Omron Sysmac Studio project MCS500_V10_2_0_Omron_EIP (Sysmac Studio 1.53.0.64009, StandardProject)
(* Mcs500 V10.2 Demo project EthernetIP *)

# Controller NX1P2_9024DT1: NX1P2-9024DT1 version 1.16
Task PrimaryTask (priority 4, period or condition 2000): MCS500_E001

TYPE MCS500 : STRUCT
    Outputs : Outputs;
    Inputs : Inputs;
    CommandsID : MCS500Cmd;
END_STRUCT END_TYPE
TYPE Inputs : STRUCT
    Status : Status;  (* offset 0.0 *)
    Motion : Motion;  (* offset 4.0 *)
    Joint_Set : Joint_Set;  (* offset 16.0 *)
    EndEffector_Pose : EndEffector_Pose;  (* offset 40.0 *)
    Configurations : Configurations;  (* offset 64.0 *)
    WRF : WRF;  (* offset 68.0 *)
    TRF : TRF;  (* offset 92.0 *)
    TimeStamp : TimeStamp;  (* offset 116.0 *)
    SafetyStatus : SafetyStatus;  (* offset 128.0 *)
    DynamicData0 : DynamicData;  (* offset 140.0 *)
    DynamicData1 : DynamicData;  (* offset 168.0 *)
    DynamicData2 : DynamicData;  (* offset 196.0 *)
    DynamicData3 : DynamicData;  (* offset 224.0 *)
END_STRUCT END_TYPE
TYPE Status : STRUCT  (* Various robot status bits *)
    Busy : BOOL;
    Activated : BOOL;
    Homed : BOOL;
    SimActivated : BOOL;
    BrakesEngaged : BOOL;
    RecoveryMode : BOOL;
    EStop : BOOL;
    CollisionStatus : BOOL;
    WorkzoneStatus : BOOL;
    Error : UINT;  (* Error code (refer to documentation for specific error code meaning) *)
END_STRUCT END_TYPE
TYPE Motion : STRUCT
    CheckPoint : UDINT;  (* Indicates which checkpoint id the robot has reached last; offset 0.0 *)
    MoveID : UINT;  (* Latest move id that was received and queued by the robot; offset 4.0 *)
    FifoSpace : UINT;  (* Number of commands that the robot can receive and queue at the moment; offset 6.0 *)
    Paused : BOOL;  (* offset 8.0 *)
    EOB : BOOL;  (* offset 8.1 *)
    EOM : BOOL;  (* offset 8.2 *)
    FifoCleared : BOOL;  (* offset 8.3 *)
    PStop2 : BOOL;  (* offset 8.4 *)
    ExcessiveTorque : BOOL;  (* offset 8.5 *)
    OfflineProgramID : UINT;  (* Id of the offline program currently running (0 if none); offset 10.0 *)
END_STRUCT END_TYPE
TYPE Joint_Set : STRUCT
    SubIndex001 : REAL;  (* Joint 1's angular position (-140 to +140) *)
    SubIndex002 : REAL;  (* Joint 2's angular position (-145 to +145) *)
    SubIndex003 : REAL;  (* Joint 3's linear position (-102 to 0) *)
    SubIndex004 : REAL;  (* Joint 4's angular position (-3600 to +3600) *)
    SubIndex005 : REAL;  (* Unused on this 4-axes robot *)
    SubIndex006 : REAL;  (* Unused on this 4-axes robot *)
END_STRUCT END_TYPE
TYPE EndEffector_Pose : STRUCT
    SubIndex001 : REAL;  (* X position *)
    SubIndex002 : REAL;  (* Y position *)
    SubIndex003 : REAL;  (* Z position *)
    SubIndex004 : REAL;  (* Alpha-angle position *)
    SubIndex005 : REAL;  (* Beta-angle position *)
    SubIndex006 : REAL;  (* Gamma-angle position *)
END_STRUCT END_TYPE
TYPE Configurations : STRUCT
    Shoulder : SINT;  (* Unused on this 4-axes robot; offset 0.0 *)
    Elbow : SINT;  (* Current elbow inverse kinematics configuration (either -1 or 1); offset 1.0 *)
    Wrist : SINT;  (* Unused on this 4-axes robot; offset 2.0 *)
    Turn : SINT;  (* Current last joint turn (-100 to 100); offset 3.0 *)
END_STRUCT END_TYPE
TYPE WRF : STRUCT
    SubIndex001 : REAL;  (* X position of WRF (relative to BRF) *)
    SubIndex002 : REAL;  (* Y position of WRF (relative to BRF) *)
    SubIndex003 : REAL;  (* Z position of WRF (relative to BRF) *)
    SubIndex004 : REAL;  (* Alpha-angle position of WRF (relative to BRF) *)
    SubIndex005 : REAL;  (* Beta-angle position of WRF (relative to BRF) *)
    SubIndex006 : REAL;  (* Gamma-angle position of WRF (relative to BRF) *)
END_STRUCT END_TYPE
TYPE TRF : STRUCT
    SubIndex001 : REAL;  (* X position of TRF (relative to FRF) *)
    SubIndex002 : REAL;  (* Y position of TRF (relative to FRF) *)
    SubIndex003 : REAL;  (* Z position of TRF (relative to FRF) *)
    SubIndex004 : REAL;  (* Alpha-angle position of TRF (relative to FRF) *)
    SubIndex005 : REAL;  (* Beta-angle position of TRF (relative to FRF) *)
    SubIndex006 : REAL;  (* Gamma-angle position of TRF (relative to FRF) *)
END_STRUCT END_TYPE
TYPE TimeStamp : STRUCT
    Seconds : UDINT;  (* Robot timestamp (seconds) indicating when input info was updated *)
    MicroSeconds : UDINT;  (* Robot timestamp (microsecond part) indicating when input info was updated *)
    DynamicDataCycles : UDINT;  (* Number of times all available dynamic data was updated *)
END_STRUCT END_TYPE
TYPE SafetyStatus : STRUCT
    EStop : BOOL;  (* offset 0.0 *)
    PStop1 : BOOL;  (* offset 0.1 *)
    PStop2 : BOOL;  (* offset 0.2 *)
    OperationModeChange : BOOL;  (* offset 0.4 *)
    EnablingDeviceReleased : BOOL;  (* offset 0.5 *)
    VoltageFluctuation : BOOL;  (* offset 0.6 *)
    Reboot : BOOL;  (* offset 0.7 *)
    RedundancyFault : BOOL;  (* offset 1.0 *)
    StandstillFault : BOOL;  (* offset 1.1 *)
    ConnectionDropped : BOOL;  (* offset 1.2 *)
    MinorError : BOOL;  (* offset 1.3 *)
    EStopResettable : BOOL;  (* offset 4.0 *)
    PStop1Resettable : BOOL;  (* offset 4.1 *)
    PStop2Resettable : BOOL;  (* offset 4.2 *)
    OperationModeChangeResettable : BOOL;  (* offset 4.4 *)
    EnablingDeviceReleasedResettable : BOOL;  (* offset 4.5 *)
    VolatgeFluctuationResettable : BOOL;  (* offset 4.6 *)
    RebootResettable : BOOL;  (* offset 4.7 *)
    RedundancyFaultResettable : BOOL;  (* offset 5.0 *)
    StandstillFaultResettable : BOOL;  (* offset 5.1 *)
    ConnectionDroppedResettable : BOOL;  (* offset 5.2 *)
    MinorErrorResettable : BOOL;  (* offset 5.3 *)
    OperationMode : SINT;  (* offset 8.0 *)
    ResetReady : BOOL;  (* offset 9.0 *)
    VMotorOn : BOOL;  (* offset 9.1 *)
    PowerSupplyInput_EStop : BOOL;  (* offset 9.2 *)
    PowerSupplyInput_PStop1 : BOOL;  (* offset 9.3 *)
    PowerSupplyInput_PStop2 : BOOL;  (* offset 9.4 *)
    PowerSupplyInput_External : BOOL;  (* offset 9.5 *)
    PowerSupplyInput_Keypad : BOOL;  (* offset 9.6 *)
    PowerSupplyInput_Enabling : BOOL;  (* offset 9.7 *)
END_STRUCT END_TYPE
TYPE DynamicData : STRUCT
    DynamicDataType : UDINT;  (* Dynamic type of the 6 following values *)
    DynamicDataValue0 : REAL;
    DynamicDataValue1 : REAL;
    DynamicDataValue2 : REAL;
    DynamicDataValue3 : REAL;
    DynamicDataValue4 : REAL;
    DynamicDataValue5 : REAL;
END_STRUCT END_TYPE
TYPE Outputs : STRUCT
    RobotControl : RobotControl;  (* offset 0.0 *)
    MotionControl : MotionControl;  (* offset 4.0 *)
    MotionCommand : MotionCommand;  (* offset 8.0 *)
    HostTime : UDINT;  (* Host absolute time in seconds since epoch (to synchronize robot's time); offset 36.0 *)
    BrakesControlAllowed : BOOL;  (* offset 40.0 *)
    BrakesEngaged : BOOL;  (* offset 40.1 *)
    DynamicDataCfg0 : UDINT;  (* Type of dynamic data to return in dynamic data index 0; offset 44.0 *)
    DynamicDataCfg1 : UDINT;  (* Type of dynamic data to return in dynamic data index 1; offset 48.0 *)
    DynamicDataCfg2 : UDINT;  (* Type of dynamic data to return in dynamic data index 2; offset 52.0 *)
    DynamicDataCfg3 : UDINT;  (* Type of dynamic data to return in dynamic data index 3; offset 56.0 *)
END_STRUCT END_TYPE
TYPE RobotControl : STRUCT  (* Various robot control bits *)
    Deactivate : BOOL;  (* offset 0.0 *)
    Activate : BOOL;  (* offset 0.1 *)
    Home : BOOL;  (* offset 0.2 *)
    ResetError : BOOL;  (* offset 0.3 *)
    EnableSimulation : BOOL;  (* offset 0.4 *)
    EnableRecoveryMode : BOOL;  (* offset 0.5 *)
    DisableEtherCAT : BOOL;  (* offset 0.6 *)
END_STRUCT END_TYPE
TYPE MotionControl : STRUCT  (* Various motion control bits *)
    MoveID : UINT;  (* User-defined id of the command currently being sent (The robot will consider a new command is sent only when moveId is changed); offset 0.0 *)
    Setpoint : BOOL;  (* offset 2.0 *)
    PauseMotion : BOOL;  (* offset 2.1 *)
    ClearMotion : BOOL;  (* offset 2.2 *)
    ResumeMotion : BOOL;  (* offset 2.3 *)
END_STRUCT END_TYPE
TYPE MotionCommand : STRUCT
    MoveCommand : UDINT;  (* The move command to apply; offset 0.0 *)
    MoveSubIndex001 : REAL;  (* Argument 1 for move command; offset 4.0 *)
    MoveSubIndex002 : REAL;  (* Argument 2 for move command; offset 8.0 *)
    MoveSubIndex003 : REAL;  (* Argument 3 for move command; offset 12.0 *)
    MoveSubIndex004 : REAL;  (* Argument 4 for move command; offset 16.0 *)
    MoveSubIndex005 : REAL;  (* Argument 5 for move command; offset 20.0 *)
    MoveSubIndex006 : REAL;  (* Argument 6 for move command; offset 24.0 *)
END_STRUCT END_TYPE
TYPE MCS500Cmd : (NoCmd := 00, MoveJoints := 01, MovePose := 02, MoveLin := 03, MoveLinRelTrf := 04, MoveLinRelWrf := 05, Delay := 06, SetBlending := 07, SetJointVel := 08, SetJointAcc := 09, SetCartAngVel := 10, SetCartLinVel := 11, SetCartAcc := 12, SetTrf := 13, SetWrf := 14, SetConf := 15, SetAutoConf := 16, SetCheckpoint := 17, MoveJointsVel := 21, MoveLinVelWrf := 22, MoveLinVelTrf := 23, SetVelTimeout := 24, SetConfTurn := 25, SetAutoConfTurn := 26, SetTorqueLimits := 27, SetTorquesLimitCfg := 28, MoveJointsRel := 29, SetJointVelLimit := 33, SetOutputState := 34, SetOutputState_Immediate := 35, SetIoSim := 36, VacuumGrip := 37, VacuumGrip_Immediate := 38, VacuumRelease := 39, VacuumRelease_Immediate := 40, SetVacuumThreshold := 41, SetVacuumThreshold_Immediate := 42, SetVacuumPurgeDuration := 43, SetVacuumPurgeDuration_Immediate := 44, MoveJump := 45, SetMoveJumpHeight := 46, SetMoveJumpApproachVel := 47, SetTimeScaling := 48, StartProgram := 100); END_TYPE

VAR_GLOBAL
    E001 : MCS500;  (* Robot Structure				PLC *)
    E001_Inputs : Inputs;  (* EthernetIp Inputs				PLC; network input *)
    E001_Outputs : Outputs;  (* EthernetIP Outputs				PLC; network output *)
END_VAR

PROGRAM MCS500_E001
VAR
    Activate : BOOL;
    Deactivate : BOOL;
    Home : BOOL;
    ResetError : BOOL;
    Pause : BOOL;
    RecoveryMode : BOOL;
    StartSequence : BOOL;
    SetCheckpoint1Buffered : BOOL;
    ExecuteMove : BOOL;
    SetCartLinVel1Buffered : BOOL;
    MovePose1Buffered : BOOL;
    SetCartLinVel1 : MCS500_SetCartLinVel;
    MovePose1 : MCS500_MovePose;
    SetCheckpoint1 : MCS500_SetCheckpoint;
    Argument : ARRAY[0..5] OF real;  (* Array for positions *)
    StepSquareMove : INT;  (* Sequencer step *)
    SetJointsVel1 : MCS500_SetJointsVel;
    SetJointsVel1Buffered : BOOL;
    ResumeMotion : BOOL;
    SetTrf1 : MCS500_SetTrf;
    SetTrf1Buffered : BOOL;
    SetWrf1 : MCS500_SetWrf;
    SetBlending1 : MCS500_SetBlending;
    SetBlending1Buffered : BOOL;
    SetConf1 : MCS500_SetConf;
    MoveLin1 : MCS500_MoveLin;
    MoveLin1Buffered : BOOL;
    SetMoveJumpApproachVel1 : MCS500_SetMoveJumpApproachVel;
    SetMoveJumpApproachVel1Buffered : BOOL;
    SetMoveJumpHeight1 : MCS500_SetMoveJumpHeight;
    SetMoveJumpHeight1Buffered : BOOL;
    MoveJump1 : MCS500_MoveJump;
    MoveJump1Buffered : BOOL;
    SetConf1Buffered : BOOL;
    E002 : MCS500;
    SetWrf1Buffered : BOOL;
    Delay1 : MCS500_Delay;
    Delay1Buffered : BOOL;
    SimulationMode : BOOL;
    ResetSequence : BOOL;
    IOModuleInfo : DWORD;
    IOModuleOutputsValues : DWORD;
    IOModuleInputsValues : DWORD;
    IOModuleSimMode : BOOL;
    IOModulePresent : BOOL;
    IOModuleErrorCode : BYTE;
    IOModuleNbInput : BYTE;
    IOModuleNbOutput : BYTE;
END_VAR
VAR_EXTERNAL
    E001_Inputs : Inputs;
    E001_Outputs : Outputs;
    E001 : MCS500;
END_VAR
VAR
    _e1 : R_TRIG;
END_VAR

(* Section IOs: ladder, written here as Structured Text *)

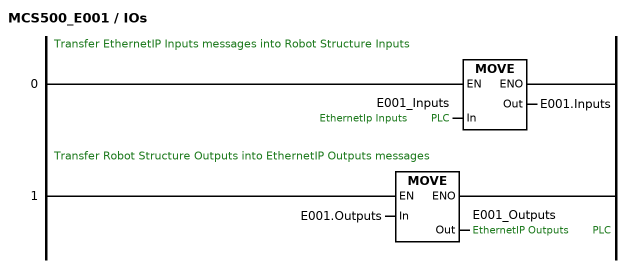
(* Rung 0: Transfer EthernetIP Inputs messages into Robot Structure Inputs *)
E001.Inputs := E001_Inputs;
(* Rung 1: Transfer Robot Structure Outputs into EthernetIP Outputs messages *)
E001_Outputs := E001.Outputs;

(* Section Robot_Control: ladder, written here as Structured Text *)

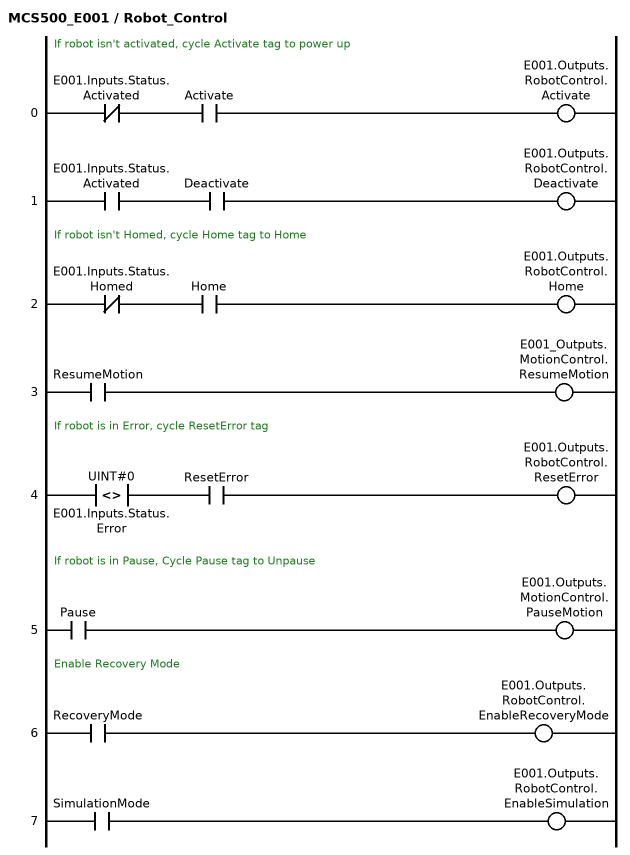
(* Rung 0: If robot isn't activated, cycle Activate tag to power up *)
E001.Outputs.RobotControl.Activate := NOT E001.Inputs.Status.Activated AND Activate;
(* Rung 1 *)
E001.Outputs.RobotControl.Deactivate := E001.Inputs.Status.Activated AND Deactivate;
(* Rung 2: If robot isn't Homed, cycle Home tag to Home *)
E001.Outputs.RobotControl.Home := NOT E001.Inputs.Status.Homed AND Home;
(* Rung 3 *)
E001_Outputs.MotionControl.ResumeMotion := ResumeMotion;
(* Rung 4: If robot is in Error, cycle ResetError tag *)
E001.Outputs.RobotControl.ResetError := (UINT#0 <> E001.Inputs.Status.Error) AND ResetError;
(* Rung 5: If robot is in Pause, Cycle Pause tag to Unpause *)
E001.Outputs.MotionControl.PauseMotion := Pause;
(* Rung 6: Enable Recovery Mode *)
E001.Outputs.RobotControl.EnableRecoveryMode := RecoveryMode;
(* Rung 7 *)
E001.Outputs.RobotControl.EnableSimulation := SimulationMode;

(* Section Sequence: ladder, written here as Structured Text *)

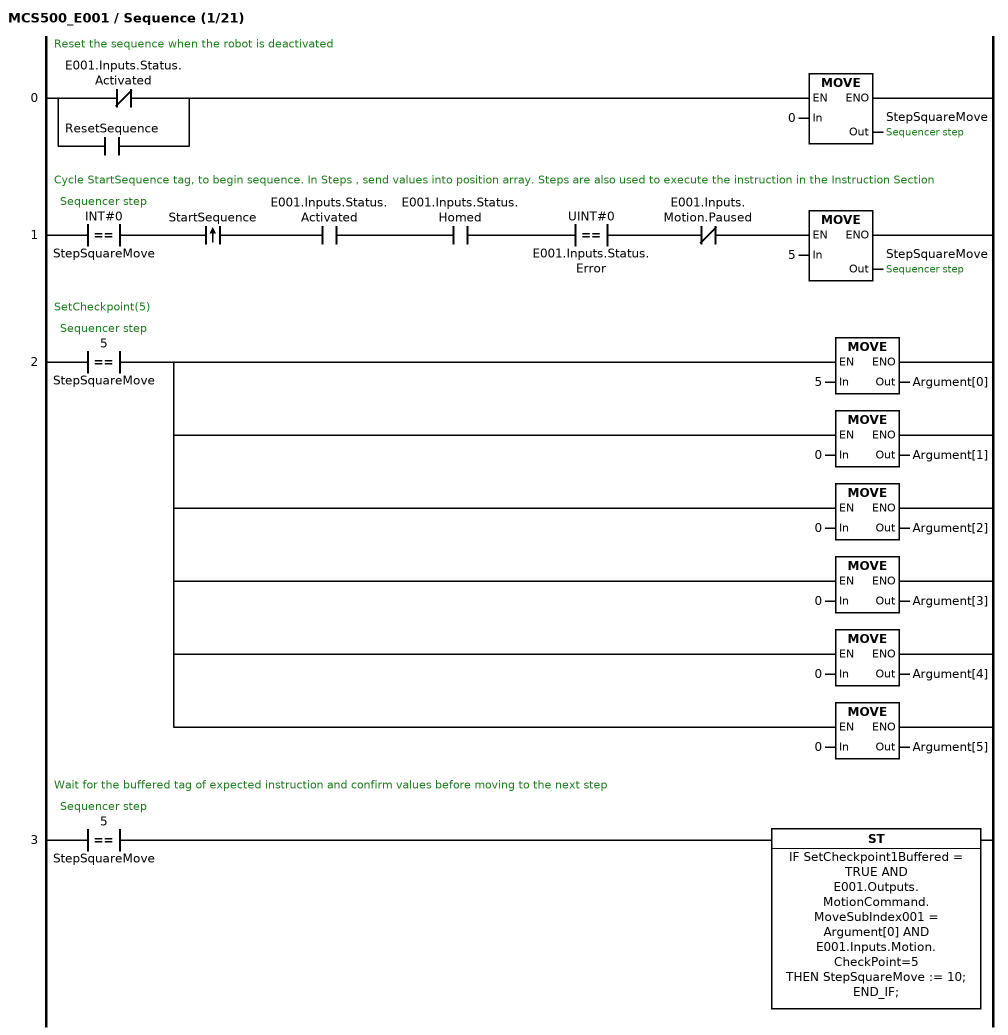
(* Rung 0: Reset the sequence when the robot is deactivated *)
IF NOT E001.Inputs.Status.Activated OR ResetSequence THEN StepSquareMove := 0; END_IF;
(* Rung 1: Cycle StartSequence tag, to begin sequence. In Steps , send values into position array. Steps are also used to execute the instruction in the Instruction Section *)
_e1(CLK := StartSequence);
IF (INT#0 = StepSquareMove) AND _e1.Q AND E001.Inputs.Status.Activated AND E001.Inputs.Status.Homed AND (UINT#0 = E001.Inputs.Status.Error) AND NOT E001.Inputs.Motion.Paused THEN
    StepSquareMove := 5;
END_IF;
(* Rung 2: SetCheckpoint(5) *)
IF 5 = StepSquareMove THEN
    Argument[0] := 5;
    Argument[1] := 0;
    Argument[2] := 0;
    Argument[3] := 0;
    Argument[4] := 0;
    Argument[5] := 0;
END_IF;
(* Rung 3: Wait for the buffered tag of expected instruction and confirm values before moving to the next step *)
IF 5 = StepSquareMove THEN
    IF SetCheckpoint1Buffered = TRUE AND
    	E001.Outputs.MotionCommand.MoveSubIndex001 = Argument[0] AND
    	E001.Inputs.Motion.CheckPoint=5
    	THEN StepSquareMove := 10;
    END_IF;
END_IF;

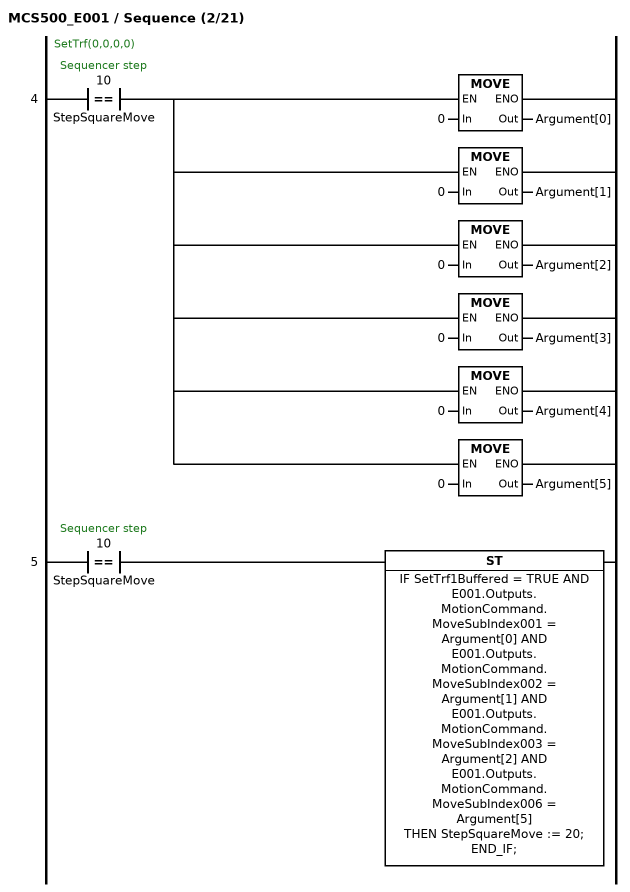
(* Rung 4: SetTrf(0,0,0,0) *)
IF 10 = StepSquareMove THEN
    Argument[0] := 0;
    Argument[1] := 0;
    Argument[2] := 0;
    Argument[3] := 0;
    Argument[4] := 0;
    Argument[5] := 0;
END_IF;
(* Rung 5 *)
IF 10 = StepSquareMove THEN
    IF SetTrf1Buffered = TRUE AND
    	E001.Outputs.MotionCommand.MoveSubIndex001 = Argument[0] AND
    	E001.Outputs.MotionCommand.MoveSubIndex002 = Argument[1] AND
    	E001.Outputs.MotionCommand.MoveSubIndex003 = Argument[2] AND
    	E001.Outputs.MotionCommand.MoveSubIndex006 = Argument[5] 
    	THEN StepSquareMove := 20;
    END_IF;
END_IF;

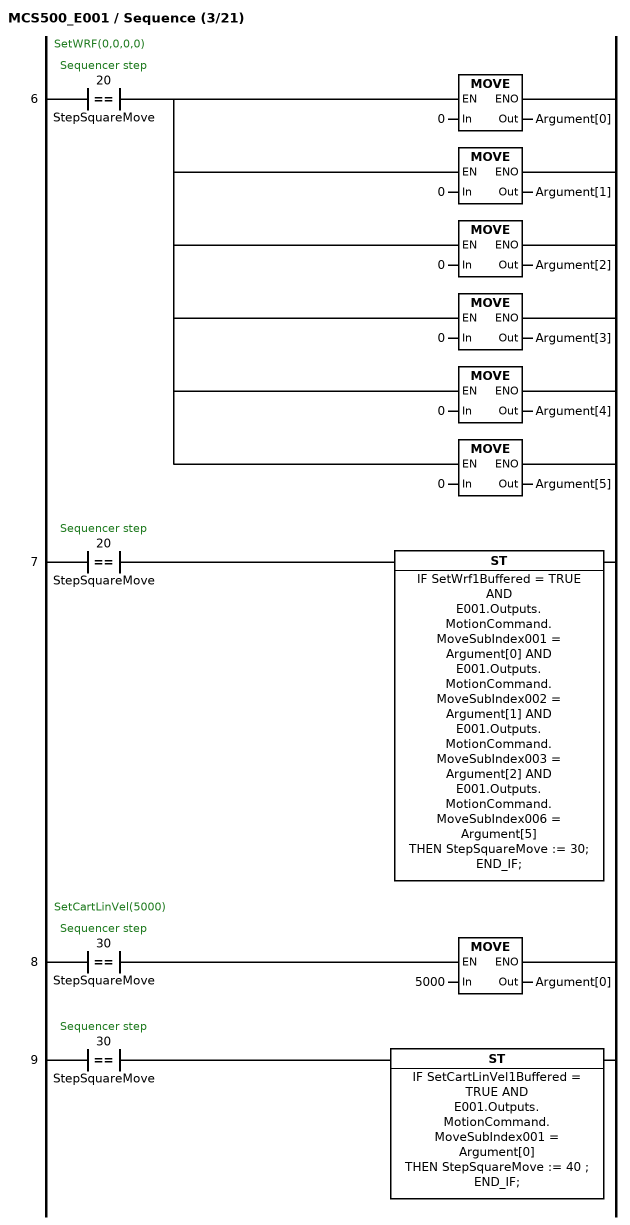
(* Rung 6: SetWRF(0,0,0,0) *)
IF 20 = StepSquareMove THEN
    Argument[0] := 0;
    Argument[1] := 0;
    Argument[2] := 0;
    Argument[3] := 0;
    Argument[4] := 0;
    Argument[5] := 0;
END_IF;
(* Rung 7 *)
IF 20 = StepSquareMove THEN
    IF SetWrf1Buffered = TRUE AND
    	E001.Outputs.MotionCommand.MoveSubIndex001 = Argument[0] AND
    	E001.Outputs.MotionCommand.MoveSubIndex002 = Argument[1] AND
    	E001.Outputs.MotionCommand.MoveSubIndex003 = Argument[2] AND
    	E001.Outputs.MotionCommand.MoveSubIndex006 = Argument[5] 
    	THEN StepSquareMove := 30;
    END_IF;
END_IF;
(* Rung 8: SetCartLinVel(5000) *)
IF 30 = StepSquareMove THEN Argument[0] := 5000; END_IF;
(* Rung 9 *)
IF 30 = StepSquareMove THEN
    IF SetCartLinVel1Buffered = TRUE AND
    	E001.Outputs.MotionCommand.MoveSubIndex001 = Argument[0] 
    	THEN StepSquareMove := 40 ;
    END_IF;
END_IF;

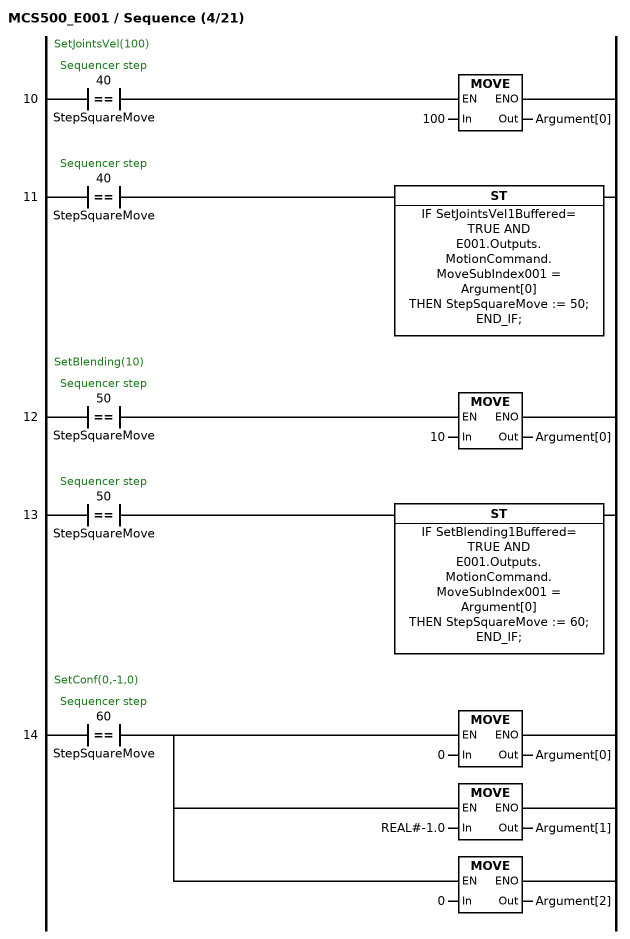
(* Rung 10: SetJointsVel(100) *)
IF 40 = StepSquareMove THEN Argument[0] := 100; END_IF;
(* Rung 11 *)
IF 40 = StepSquareMove THEN
    IF SetJointsVel1Buffered= TRUE AND
    	E001.Outputs.MotionCommand.MoveSubIndex001 = Argument[0]
    	THEN StepSquareMove := 50;
    END_IF;
END_IF;
(* Rung 12: SetBlending(10) *)
IF 50 = StepSquareMove THEN Argument[0] := 10; END_IF;
(* Rung 13 *)
IF 50 = StepSquareMove THEN
    IF SetBlending1Buffered= TRUE AND
    	E001.Outputs.MotionCommand.MoveSubIndex001 = Argument[0]
    	THEN StepSquareMove := 60;
    END_IF;
END_IF;
(* Rung 14: SetConf(0,-1,0) *)
IF 60 = StepSquareMove THEN
    Argument[0] := 0;
    Argument[1] := REAL#-1.0;
    Argument[2] := 0;
END_IF;

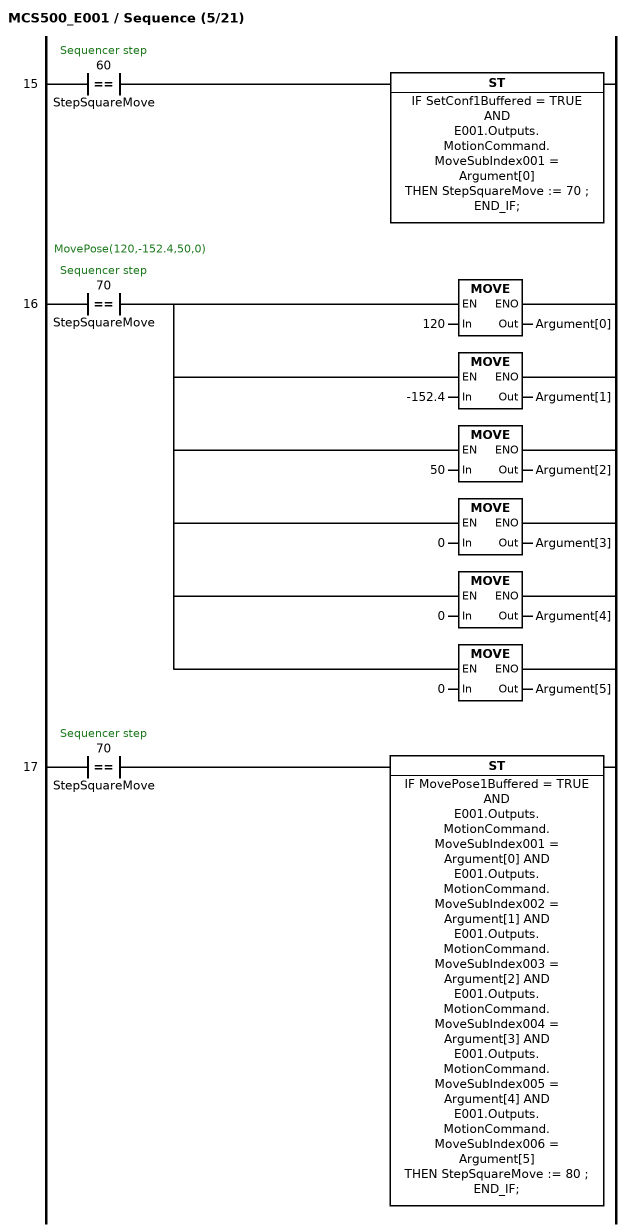
(* Rung 15 *)
IF 60 = StepSquareMove THEN
    IF SetConf1Buffered = TRUE AND
    	E001.Outputs.MotionCommand.MoveSubIndex001 = Argument[0]
    	THEN StepSquareMove := 70 ;
    END_IF;
END_IF;
(* Rung 16: MovePose(120,-152.4,50,0) *)
IF 70 = StepSquareMove THEN
    Argument[0] := 120;
    Argument[1] := -152.4;
    Argument[2] := 50;
    Argument[3] := 0;
    Argument[4] := 0;
    Argument[5] := 0;
END_IF;
(* Rung 17 *)
IF 70 = StepSquareMove THEN
    IF MovePose1Buffered = TRUE AND
    	E001.Outputs.MotionCommand.MoveSubIndex001 = Argument[0] AND
    	E001.Outputs.MotionCommand.MoveSubIndex002 = Argument[1] AND
    	E001.Outputs.MotionCommand.MoveSubIndex003 = Argument[2] AND
    	E001.Outputs.MotionCommand.MoveSubIndex004 = Argument[3] AND
    	E001.Outputs.MotionCommand.MoveSubIndex005 = Argument[4] AND
    	E001.Outputs.MotionCommand.MoveSubIndex006 = Argument[5] 
    	THEN StepSquareMove := 80 ;
    END_IF;
END_IF;

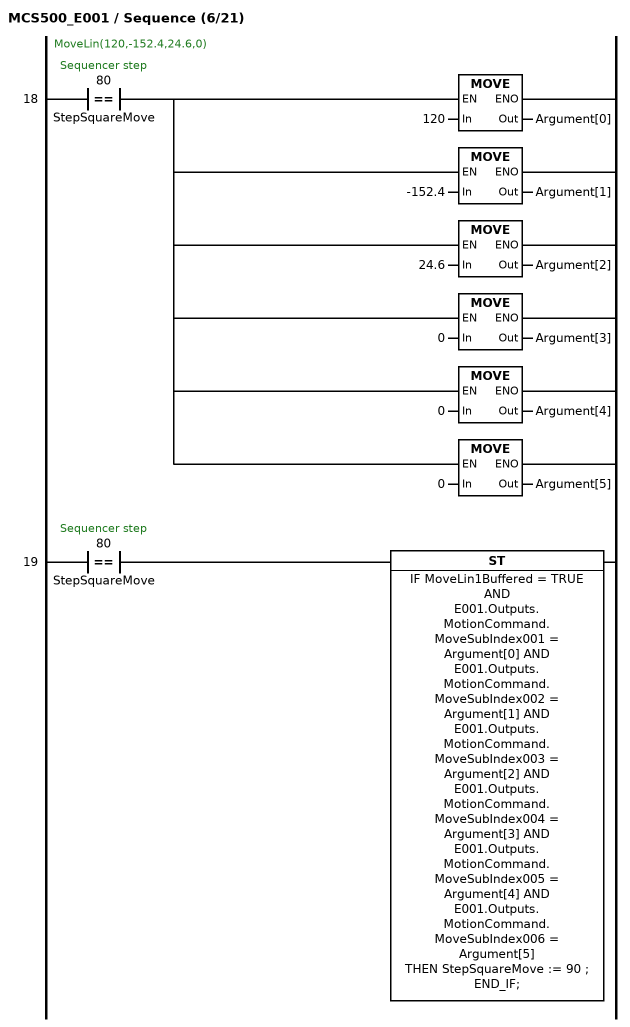
(* Rung 18: MoveLin(120,-152.4,24.6,0) *)
IF 80 = StepSquareMove THEN
    Argument[0] := 120;
    Argument[1] := -152.4;
    Argument[2] := 24.6;
    Argument[3] := 0;
    Argument[4] := 0;
    Argument[5] := 0;
END_IF;
(* Rung 19 *)
IF 80 = StepSquareMove THEN
    IF MoveLin1Buffered = TRUE AND
    	E001.Outputs.MotionCommand.MoveSubIndex001 = Argument[0] AND
    	E001.Outputs.MotionCommand.MoveSubIndex002 = Argument[1] AND
    	E001.Outputs.MotionCommand.MoveSubIndex003 = Argument[2] AND
    	E001.Outputs.MotionCommand.MoveSubIndex004 = Argument[3] AND
    	E001.Outputs.MotionCommand.MoveSubIndex005 = Argument[4] AND
    	E001.Outputs.MotionCommand.MoveSubIndex006 = Argument[5] 
    	THEN StepSquareMove := 90 ;
    END_IF;
END_IF;

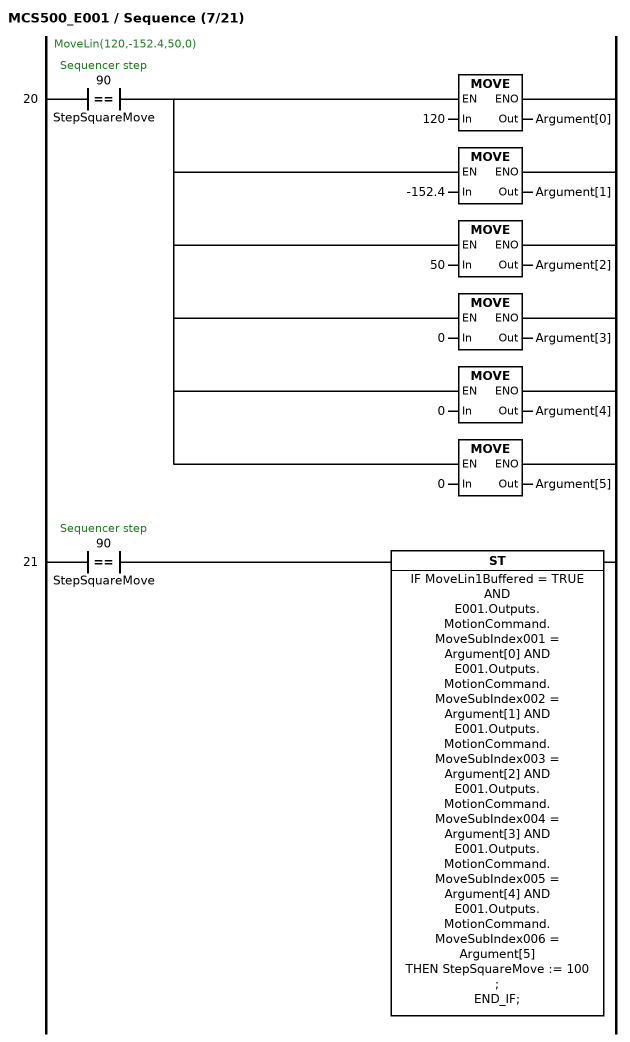
(* Rung 20: MoveLin(120,-152.4,50,0) *)
IF 90 = StepSquareMove THEN
    Argument[0] := 120;
    Argument[1] := -152.4;
    Argument[2] := 50;
    Argument[3] := 0;
    Argument[4] := 0;
    Argument[5] := 0;
END_IF;
(* Rung 21 *)
IF 90 = StepSquareMove THEN
    IF MoveLin1Buffered = TRUE AND
    	E001.Outputs.MotionCommand.MoveSubIndex001 = Argument[0] AND
    	E001.Outputs.MotionCommand.MoveSubIndex002 = Argument[1] AND
    	E001.Outputs.MotionCommand.MoveSubIndex003 = Argument[2] AND
    	E001.Outputs.MotionCommand.MoveSubIndex004 = Argument[3] AND
    	E001.Outputs.MotionCommand.MoveSubIndex005 = Argument[4] AND
    	E001.Outputs.MotionCommand.MoveSubIndex006 = Argument[5] 
    	THEN StepSquareMove := 100 ;
    END_IF;
END_IF;

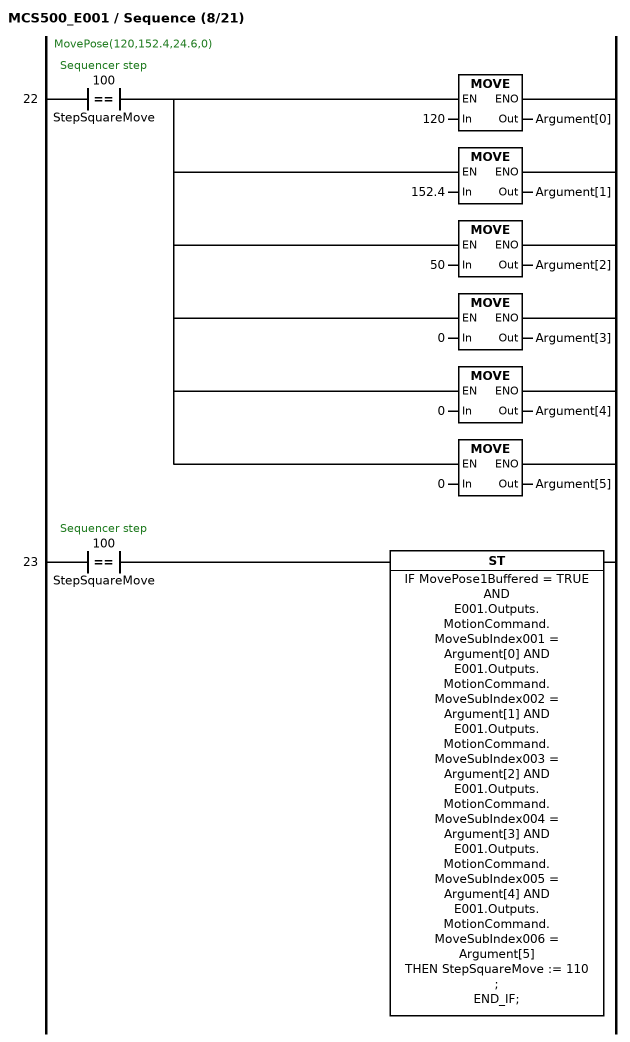
(* Rung 22: MovePose(120,152.4,24.6,0) *)
IF 100 = StepSquareMove THEN
    Argument[0] := 120;
    Argument[1] := 152.4;
    Argument[2] := 50;
    Argument[3] := 0;
    Argument[4] := 0;
    Argument[5] := 0;
END_IF;
(* Rung 23 *)
IF 100 = StepSquareMove THEN
    IF MovePose1Buffered = TRUE AND
    	E001.Outputs.MotionCommand.MoveSubIndex001 = Argument[0] AND
    	E001.Outputs.MotionCommand.MoveSubIndex002 = Argument[1] AND
    	E001.Outputs.MotionCommand.MoveSubIndex003 = Argument[2] AND
    	E001.Outputs.MotionCommand.MoveSubIndex004 = Argument[3] AND
    	E001.Outputs.MotionCommand.MoveSubIndex005 = Argument[4] AND
    	E001.Outputs.MotionCommand.MoveSubIndex006 = Argument[5] 
    	THEN StepSquareMove := 110 ;
    END_IF;
END_IF;

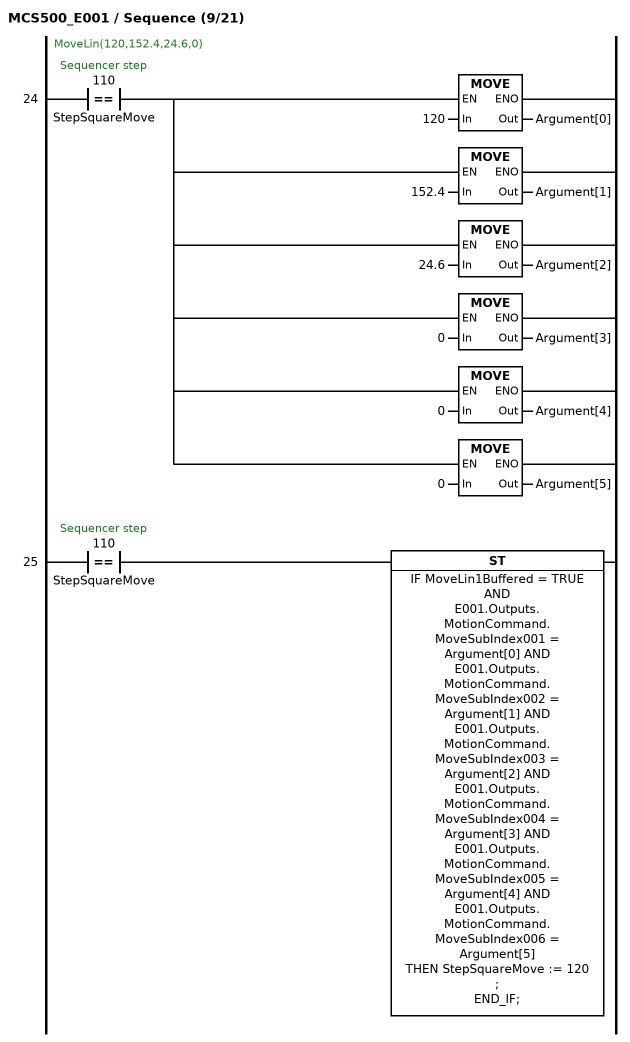
(* Rung 24: MoveLin(120,152.4,24.6,0) *)
IF 110 = StepSquareMove THEN
    Argument[0] := 120;
    Argument[1] := 152.4;
    Argument[2] := 24.6;
    Argument[3] := 0;
    Argument[4] := 0;
    Argument[5] := 0;
END_IF;
(* Rung 25 *)
IF 110 = StepSquareMove THEN
    IF MoveLin1Buffered = TRUE AND
    	E001.Outputs.MotionCommand.MoveSubIndex001 = Argument[0] AND
    	E001.Outputs.MotionCommand.MoveSubIndex002 = Argument[1] AND
    	E001.Outputs.MotionCommand.MoveSubIndex003 = Argument[2] AND
    	E001.Outputs.MotionCommand.MoveSubIndex004 = Argument[3] AND
    	E001.Outputs.MotionCommand.MoveSubIndex005 = Argument[4] AND
    	E001.Outputs.MotionCommand.MoveSubIndex006 = Argument[5] 
    	THEN StepSquareMove := 120 ;
    END_IF;
END_IF;

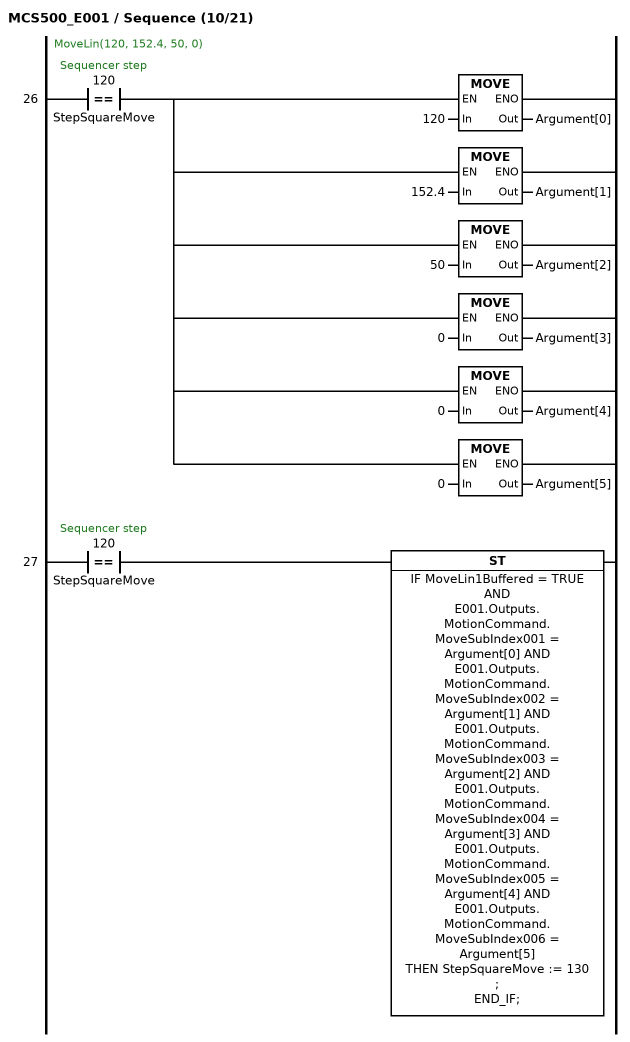
(* Rung 26: MoveLin(120, 152.4, 50, 0) *)
IF 120 = StepSquareMove THEN
    Argument[0] := 120;
    Argument[1] := 152.4;
    Argument[2] := 50;
    Argument[3] := 0;
    Argument[4] := 0;
    Argument[5] := 0;
END_IF;
(* Rung 27 *)
IF 120 = StepSquareMove THEN
    IF MoveLin1Buffered = TRUE AND
    	E001.Outputs.MotionCommand.MoveSubIndex001 = Argument[0] AND
    	E001.Outputs.MotionCommand.MoveSubIndex002 = Argument[1] AND
    	E001.Outputs.MotionCommand.MoveSubIndex003 = Argument[2] AND
    	E001.Outputs.MotionCommand.MoveSubIndex004 = Argument[3] AND
    	E001.Outputs.MotionCommand.MoveSubIndex005 = Argument[4] AND
    	E001.Outputs.MotionCommand.MoveSubIndex006 = Argument[5] 
    	THEN StepSquareMove := 130 ;
    END_IF;
END_IF;

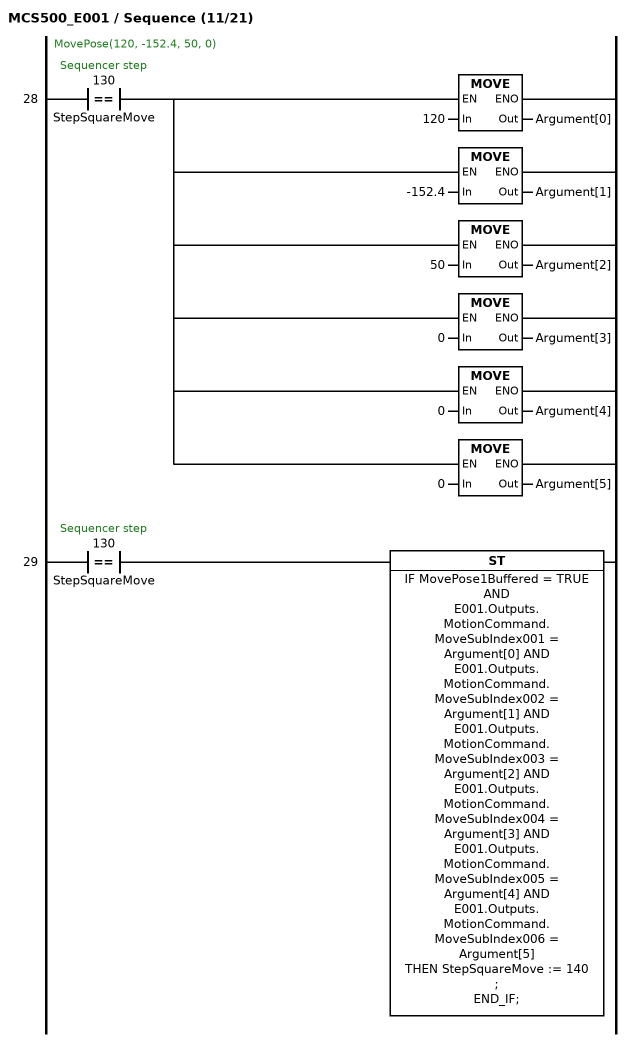
(* Rung 28: MovePose(120, -152.4, 50, 0) *)
IF 130 = StepSquareMove THEN
    Argument[0] := 120;
    Argument[1] := -152.4;
    Argument[2] := 50;
    Argument[3] := 0;
    Argument[4] := 0;
    Argument[5] := 0;
END_IF;
(* Rung 29 *)
IF 130 = StepSquareMove THEN
    IF MovePose1Buffered = TRUE AND
    	E001.Outputs.MotionCommand.MoveSubIndex001 = Argument[0] AND
    	E001.Outputs.MotionCommand.MoveSubIndex002 = Argument[1] AND
    	E001.Outputs.MotionCommand.MoveSubIndex003 = Argument[2] AND
    	E001.Outputs.MotionCommand.MoveSubIndex004 = Argument[3] AND
    	E001.Outputs.MotionCommand.MoveSubIndex005 = Argument[4] AND
    	E001.Outputs.MotionCommand.MoveSubIndex006 = Argument[5] 
    	THEN StepSquareMove := 140 ;
    END_IF;
END_IF;

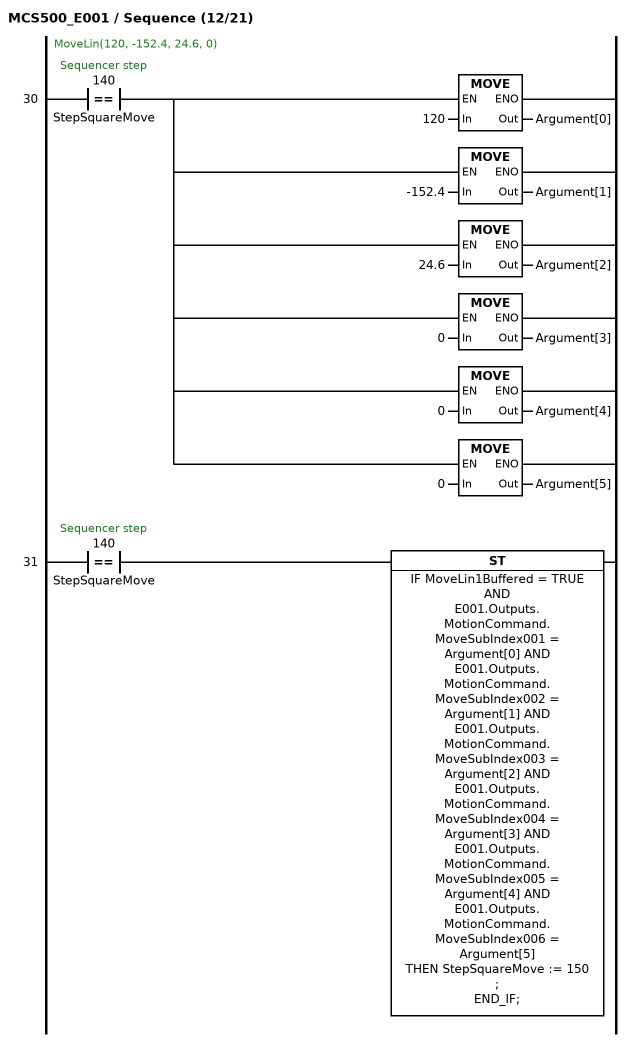
(* Rung 30: MoveLin(120, -152.4, 24.6, 0) *)
IF 140 = StepSquareMove THEN
    Argument[0] := 120;
    Argument[1] := -152.4;
    Argument[2] := 24.6;
    Argument[3] := 0;
    Argument[4] := 0;
    Argument[5] := 0;
END_IF;
(* Rung 31 *)
IF 140 = StepSquareMove THEN
    IF MoveLin1Buffered = TRUE AND
    	E001.Outputs.MotionCommand.MoveSubIndex001 = Argument[0] AND
    	E001.Outputs.MotionCommand.MoveSubIndex002 = Argument[1] AND
    	E001.Outputs.MotionCommand.MoveSubIndex003 = Argument[2] AND
    	E001.Outputs.MotionCommand.MoveSubIndex004 = Argument[3] AND
    	E001.Outputs.MotionCommand.MoveSubIndex005 = Argument[4] AND
    	E001.Outputs.MotionCommand.MoveSubIndex006 = Argument[5] 
    	THEN StepSquareMove := 150 ;
    END_IF;
END_IF;

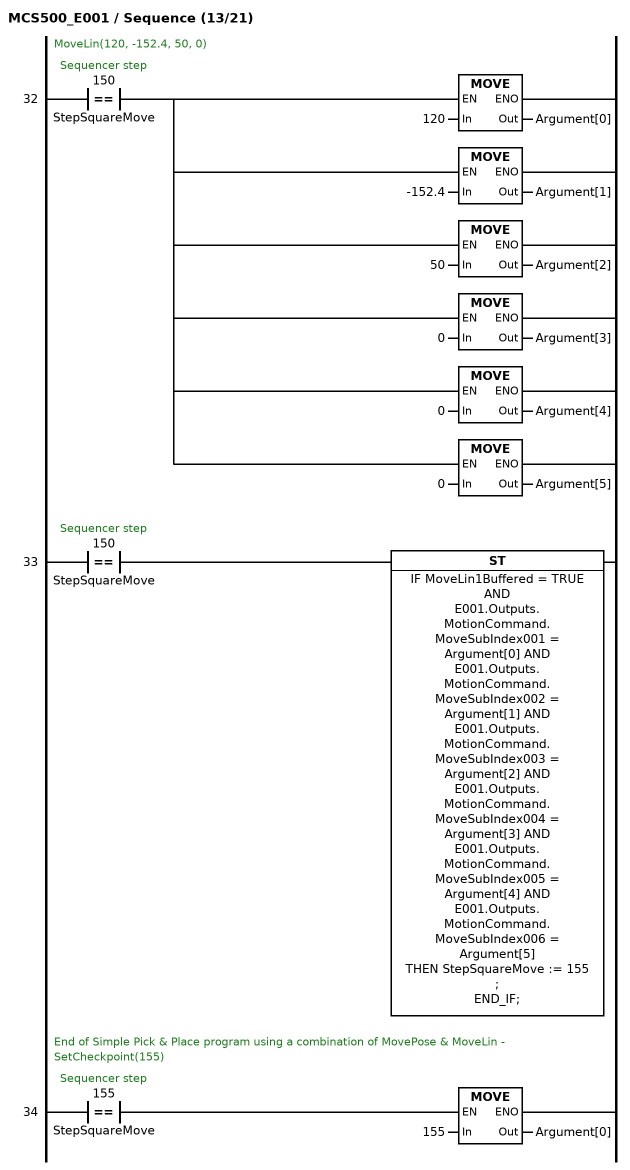
(* Rung 32: MoveLin(120, -152.4, 50, 0) *)
IF 150 = StepSquareMove THEN
    Argument[0] := 120;
    Argument[1] := -152.4;
    Argument[2] := 50;
    Argument[3] := 0;
    Argument[4] := 0;
    Argument[5] := 0;
END_IF;
(* Rung 33 *)
IF 150 = StepSquareMove THEN
    IF MoveLin1Buffered = TRUE AND
    	E001.Outputs.MotionCommand.MoveSubIndex001 = Argument[0] AND
    	E001.Outputs.MotionCommand.MoveSubIndex002 = Argument[1] AND
    	E001.Outputs.MotionCommand.MoveSubIndex003 = Argument[2] AND
    	E001.Outputs.MotionCommand.MoveSubIndex004 = Argument[3] AND
    	E001.Outputs.MotionCommand.MoveSubIndex005 = Argument[4] AND
    	E001.Outputs.MotionCommand.MoveSubIndex006 = Argument[5] 
    	THEN StepSquareMove := 155 ;
    END_IF;
END_IF;
(* Rung 34: End of Simple Pick & Place program using a combination of MovePose & MoveLin - SetCheckpoint(155) *)
IF 155 = StepSquareMove THEN Argument[0] := 155; END_IF;

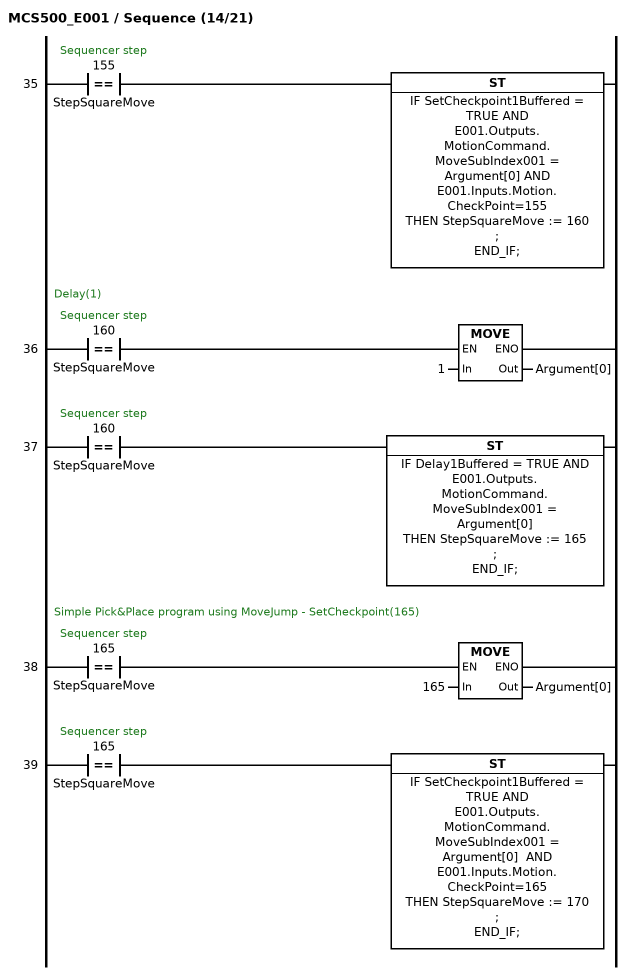
(* Rung 35 *)
IF 155 = StepSquareMove THEN
    IF SetCheckpoint1Buffered = TRUE AND
    	E001.Outputs.MotionCommand.MoveSubIndex001 = Argument[0] AND
    	E001.Inputs.Motion.CheckPoint=155
    	THEN StepSquareMove := 160 ;
    END_IF;
END_IF;
(* Rung 36: Delay(1) *)
IF 160 = StepSquareMove THEN Argument[0] := 1; END_IF;
(* Rung 37 *)
IF 160 = StepSquareMove THEN
    IF Delay1Buffered = TRUE AND
    	E001.Outputs.MotionCommand.MoveSubIndex001 = Argument[0]  
    	THEN StepSquareMove := 165 ;
    END_IF;
END_IF;
(* Rung 38: Simple Pick&Place program using MoveJump - SetCheckpoint(165) *)
IF 165 = StepSquareMove THEN Argument[0] := 165; END_IF;
(* Rung 39 *)
IF 165 = StepSquareMove THEN
    IF SetCheckpoint1Buffered = TRUE AND
    	E001.Outputs.MotionCommand.MoveSubIndex001 = Argument[0]  AND
    	E001.Inputs.Motion.CheckPoint=165
    	THEN StepSquareMove := 170 ;
    END_IF;
END_IF;

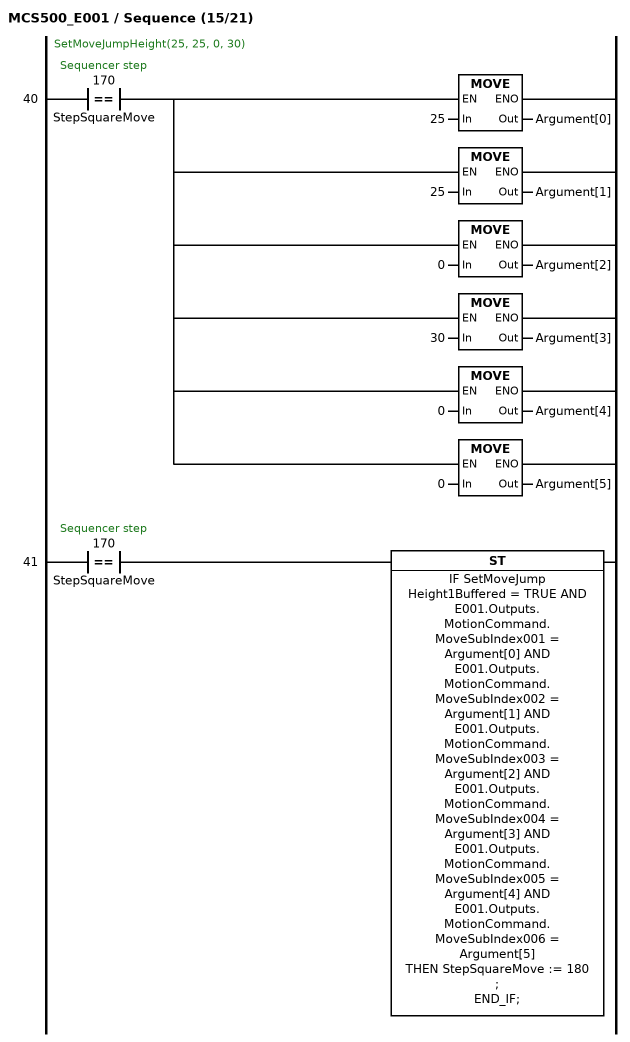
(* Rung 40: SetMoveJumpHeight(25, 25, 0, 30) *)
IF 170 = StepSquareMove THEN
    Argument[0] := 25;
    Argument[1] := 25;
    Argument[2] := 0;
    Argument[3] := 30;
    Argument[4] := 0;
    Argument[5] := 0;
END_IF;
(* Rung 41 *)
IF 170 = StepSquareMove THEN
    IF SetMoveJumpHeight1Buffered = TRUE AND
    	E001.Outputs.MotionCommand.MoveSubIndex001 = Argument[0] AND
    	E001.Outputs.MotionCommand.MoveSubIndex002 = Argument[1] AND
    	E001.Outputs.MotionCommand.MoveSubIndex003 = Argument[2] AND
    	E001.Outputs.MotionCommand.MoveSubIndex004 = Argument[3] AND
    	E001.Outputs.MotionCommand.MoveSubIndex005 = Argument[4] AND
    	E001.Outputs.MotionCommand.MoveSubIndex006 = Argument[5] 
    	THEN StepSquareMove := 180 ;
    END_IF;
END_IF;

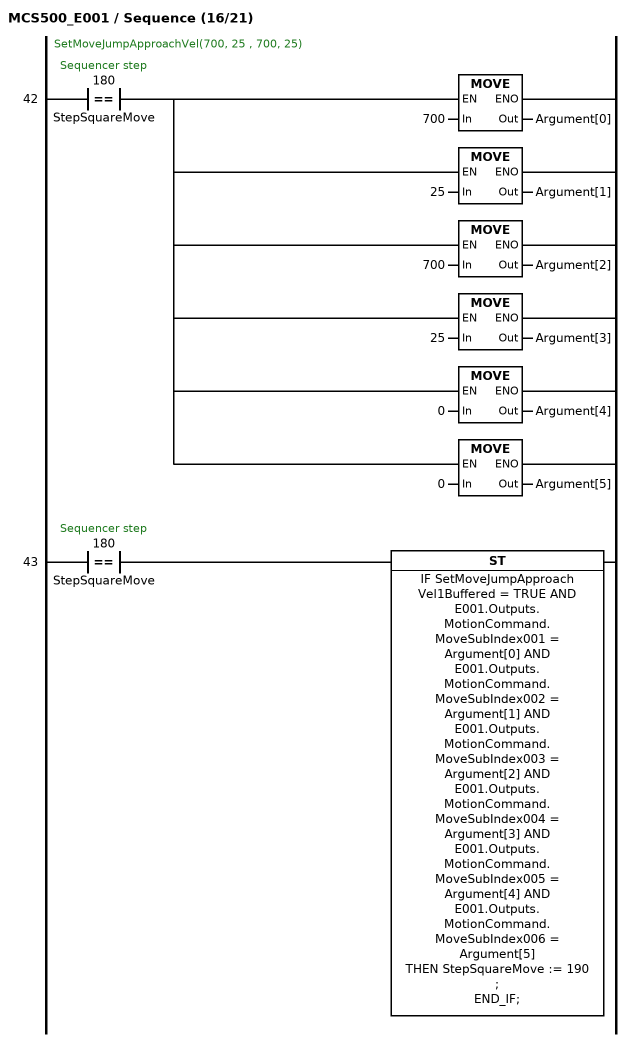
(* Rung 42: SetMoveJumpApproachVel(700, 25 , 700, 25) *)
IF 180 = StepSquareMove THEN
    Argument[0] := 700;
    Argument[1] := 25;
    Argument[2] := 700;
    Argument[3] := 25;
    Argument[4] := 0;
    Argument[5] := 0;
END_IF;
(* Rung 43 *)
IF 180 = StepSquareMove THEN
    IF SetMoveJumpApproachVel1Buffered = TRUE AND
    	E001.Outputs.MotionCommand.MoveSubIndex001 = Argument[0] AND
    	E001.Outputs.MotionCommand.MoveSubIndex002 = Argument[1] AND
    	E001.Outputs.MotionCommand.MoveSubIndex003 = Argument[2] AND
    	E001.Outputs.MotionCommand.MoveSubIndex004 = Argument[3] AND
    	E001.Outputs.MotionCommand.MoveSubIndex005 = Argument[4] AND
    	E001.Outputs.MotionCommand.MoveSubIndex006 = Argument[5] 
    	THEN StepSquareMove := 190 ;
    END_IF;
END_IF;

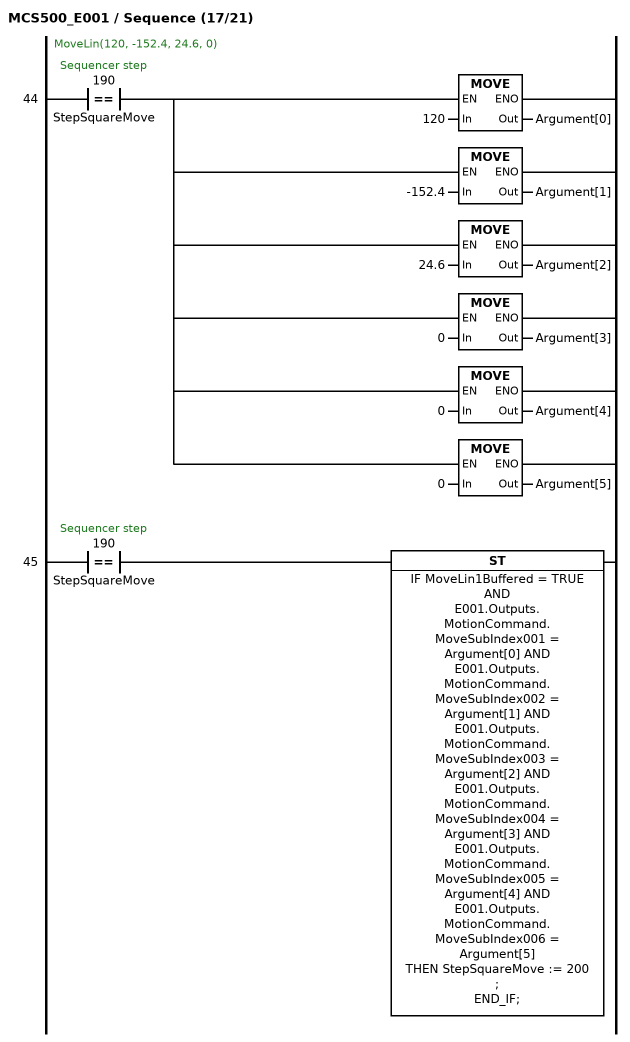
(* Rung 44: MoveLin(120, -152.4, 24.6, 0) *)
IF 190 = StepSquareMove THEN
    Argument[0] := 120;
    Argument[1] := -152.4;
    Argument[2] := 24.6;
    Argument[3] := 0;
    Argument[4] := 0;
    Argument[5] := 0;
END_IF;
(* Rung 45 *)
IF 190 = StepSquareMove THEN
    IF MoveLin1Buffered = TRUE AND
    	E001.Outputs.MotionCommand.MoveSubIndex001 = Argument[0] AND
    	E001.Outputs.MotionCommand.MoveSubIndex002 = Argument[1] AND
    	E001.Outputs.MotionCommand.MoveSubIndex003 = Argument[2] AND
    	E001.Outputs.MotionCommand.MoveSubIndex004 = Argument[3] AND
    	E001.Outputs.MotionCommand.MoveSubIndex005 = Argument[4] AND
    	E001.Outputs.MotionCommand.MoveSubIndex006 = Argument[5] 
    	THEN StepSquareMove := 200 ;
    END_IF;
END_IF;

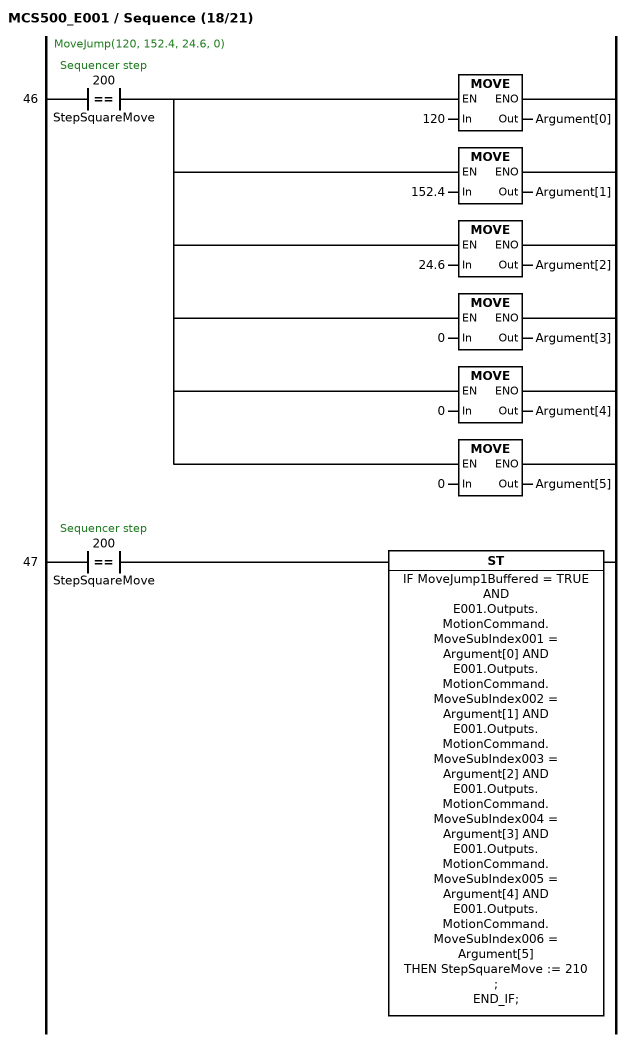
(* Rung 46: MoveJump(120, 152.4, 24.6, 0) *)
IF 200 = StepSquareMove THEN
    Argument[0] := 120;
    Argument[1] := 152.4;
    Argument[2] := 24.6;
    Argument[3] := 0;
    Argument[4] := 0;
    Argument[5] := 0;
END_IF;
(* Rung 47 *)
IF 200 = StepSquareMove THEN
    IF MoveJump1Buffered = TRUE AND
    	E001.Outputs.MotionCommand.MoveSubIndex001 = Argument[0] AND
    	E001.Outputs.MotionCommand.MoveSubIndex002 = Argument[1] AND
    	E001.Outputs.MotionCommand.MoveSubIndex003 = Argument[2] AND
    	E001.Outputs.MotionCommand.MoveSubIndex004 = Argument[3] AND
    	E001.Outputs.MotionCommand.MoveSubIndex005 = Argument[4] AND
    	E001.Outputs.MotionCommand.MoveSubIndex006 = Argument[5] 
    	THEN StepSquareMove := 210 ;
    END_IF;
END_IF;

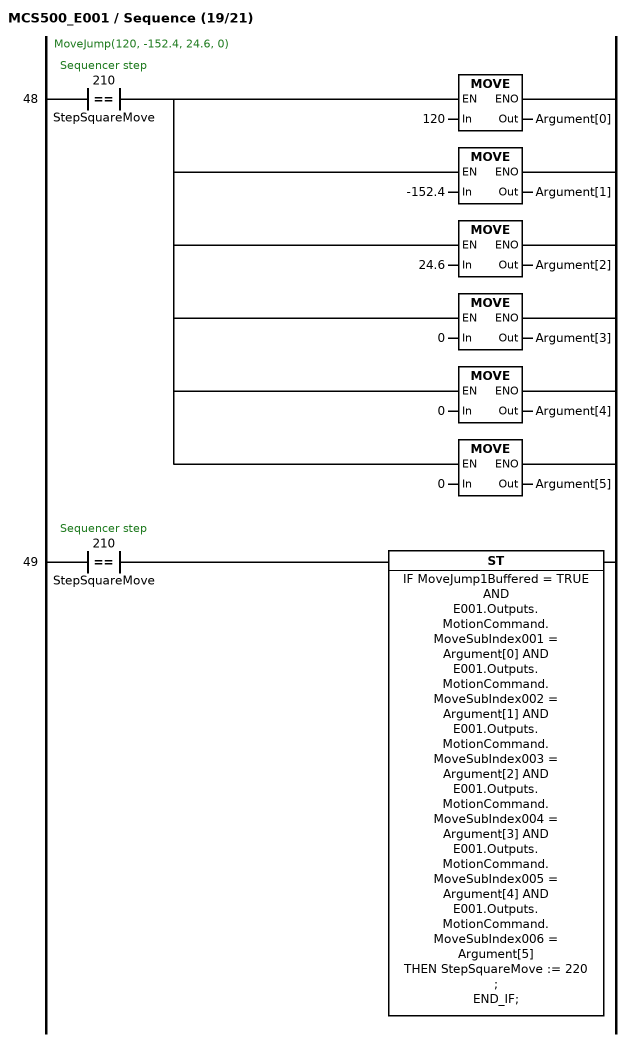
(* Rung 48: MoveJump(120, -152.4, 24.6, 0) *)
IF 210 = StepSquareMove THEN
    Argument[0] := 120;
    Argument[1] := -152.4;
    Argument[2] := 24.6;
    Argument[3] := 0;
    Argument[4] := 0;
    Argument[5] := 0;
END_IF;
(* Rung 49 *)
IF 210 = StepSquareMove THEN
    IF MoveJump1Buffered = TRUE AND
    	E001.Outputs.MotionCommand.MoveSubIndex001 = Argument[0] AND
    	E001.Outputs.MotionCommand.MoveSubIndex002 = Argument[1] AND
    	E001.Outputs.MotionCommand.MoveSubIndex003 = Argument[2] AND
    	E001.Outputs.MotionCommand.MoveSubIndex004 = Argument[3] AND
    	E001.Outputs.MotionCommand.MoveSubIndex005 = Argument[4] AND
    	E001.Outputs.MotionCommand.MoveSubIndex006 = Argument[5] 
    	THEN StepSquareMove := 220 ;
    END_IF;
END_IF;

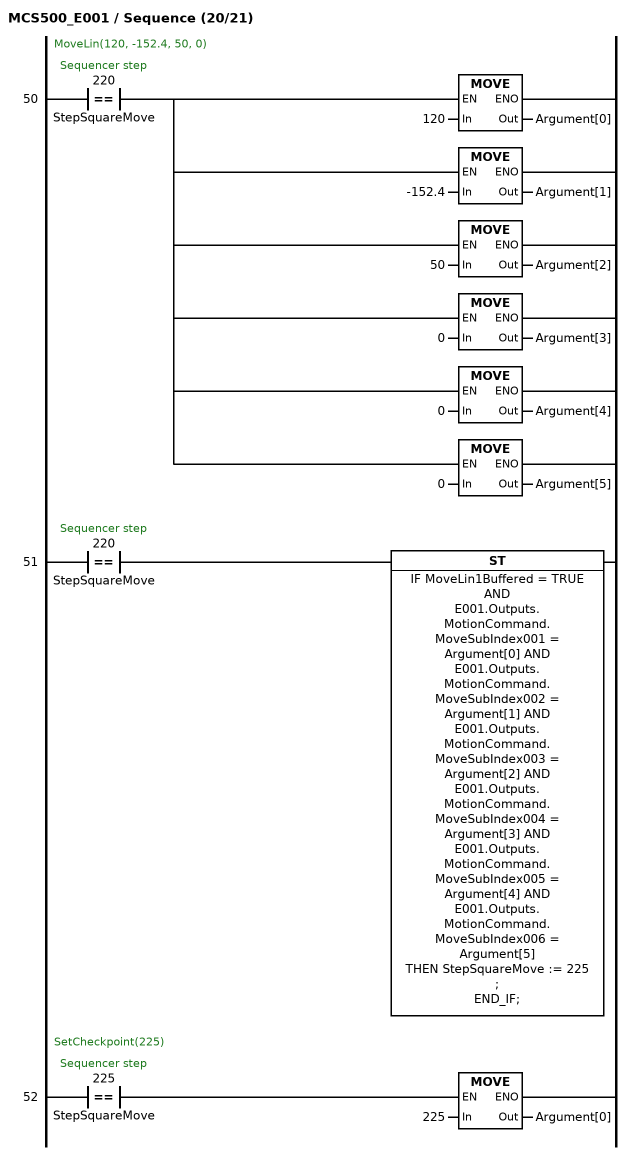
(* Rung 50: MoveLin(120, -152.4, 50, 0) *)
IF 220 = StepSquareMove THEN
    Argument[0] := 120;
    Argument[1] := -152.4;
    Argument[2] := 50;
    Argument[3] := 0;
    Argument[4] := 0;
    Argument[5] := 0;
END_IF;
(* Rung 51 *)
IF 220 = StepSquareMove THEN
    IF MoveLin1Buffered = TRUE AND
    	E001.Outputs.MotionCommand.MoveSubIndex001 = Argument[0] AND
    	E001.Outputs.MotionCommand.MoveSubIndex002 = Argument[1] AND
    	E001.Outputs.MotionCommand.MoveSubIndex003 = Argument[2] AND
    	E001.Outputs.MotionCommand.MoveSubIndex004 = Argument[3] AND
    	E001.Outputs.MotionCommand.MoveSubIndex005 = Argument[4] AND
    	E001.Outputs.MotionCommand.MoveSubIndex006 = Argument[5] 
    	THEN StepSquareMove := 225 ;
    END_IF;
END_IF;
(* Rung 52: SetCheckpoint(225) *)
IF 225 = StepSquareMove THEN Argument[0] := 225; END_IF;

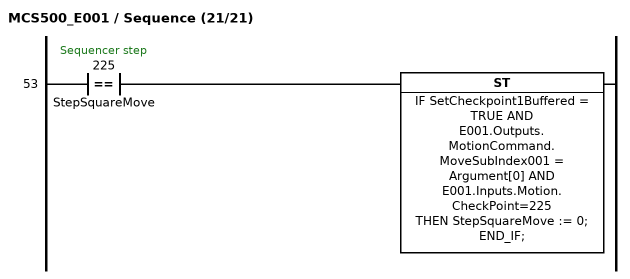
(* Rung 53 *)
IF 225 = StepSquareMove THEN
    IF SetCheckpoint1Buffered = TRUE AND
    	E001.Outputs.MotionCommand.MoveSubIndex001 = Argument[0] AND
    	E001.Inputs.Motion.CheckPoint=225
    	THEN StepSquareMove := 0;
    END_IF;
END_IF;

(* Section Instructions: ladder, written here as Structured Text *)

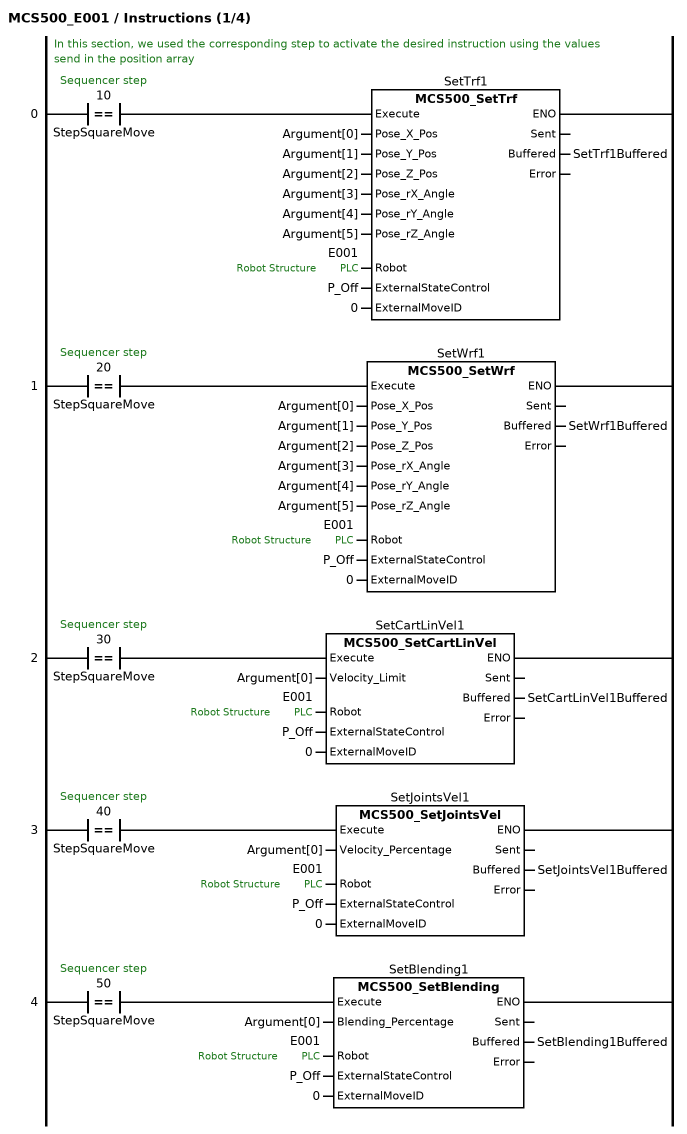
(* Rung 0: In this section, we used the corresponding step to activate the desired instruction using the values send in the position array *)
SetTrf1(Execute := 10 = StepSquareMove, Pose_X_Pos := Argument[0], Pose_Y_Pos := Argument[1], Pose_Z_Pos := Argument[2], Pose_rX_Angle := Argument[3], Pose_rY_Angle := Argument[4], Pose_rZ_Angle := Argument[5], Robot := E001, ExternalStateControl := P_Off, ExternalMoveID := 0, Buffered => SetTrf1Buffered);
(* Rung 1 *)
SetWrf1(Execute := 20 = StepSquareMove, Pose_X_Pos := Argument[0], Pose_Y_Pos := Argument[1], Pose_Z_Pos := Argument[2], Pose_rX_Angle := Argument[3], Pose_rY_Angle := Argument[4], Pose_rZ_Angle := Argument[5], Robot := E001, ExternalStateControl := P_Off, ExternalMoveID := 0, Buffered => SetWrf1Buffered);
(* Rung 2 *)
SetCartLinVel1(Execute := 30 = StepSquareMove, Velocity_Limit := Argument[0], Robot := E001, ExternalStateControl := P_Off, ExternalMoveID := 0, Buffered => SetCartLinVel1Buffered);
(* Rung 3 *)
SetJointsVel1(Execute := 40 = StepSquareMove, Velocity_Percentage := Argument[0], Robot := E001, ExternalStateControl := P_Off, ExternalMoveID := 0, Buffered => SetJointsVel1Buffered);
(* Rung 4 *)
SetBlending1(Execute := 50 = StepSquareMove, Blending_Percentage := Argument[0], Robot := E001, ExternalStateControl := P_Off, ExternalMoveID := 0, Buffered => SetBlending1Buffered);

